FUNCTION_BLOCK GripperCtrl (* Template for a simple Basic Function Block Type *)
  (* Standard: 61499-2 *)
  (* Version 1.0, 2018-07-09, az *)
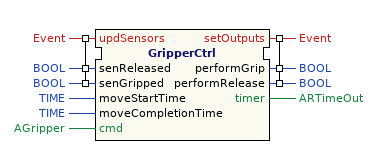
  EVENT_INPUT
    updSensors WITH senReleased, senGripped;
  END_EVENT
  EVENT_OUTPUT
    setOutputs WITH performGrip, performRelease;
  END_EVENT
  VAR_INPUT
    senReleased : BOOL;
    senGripped : BOOL;
    moveStartTime : TIME; (* timeout value till a move should start *)
    moveCompletionTime : TIME; (* timeout till a full movement completes *)
  END_VAR
  VAR_OUTPUT
    performGrip : BOOL;
    performRelease : BOOL;
  END_VAR
  SOCKETS
    cmd : AGripper; (* Command interface for requesting gripper actions *)
  END_SOCKETS
  PLUGS
    timer : ARTimeOut;
  END_PLUGS
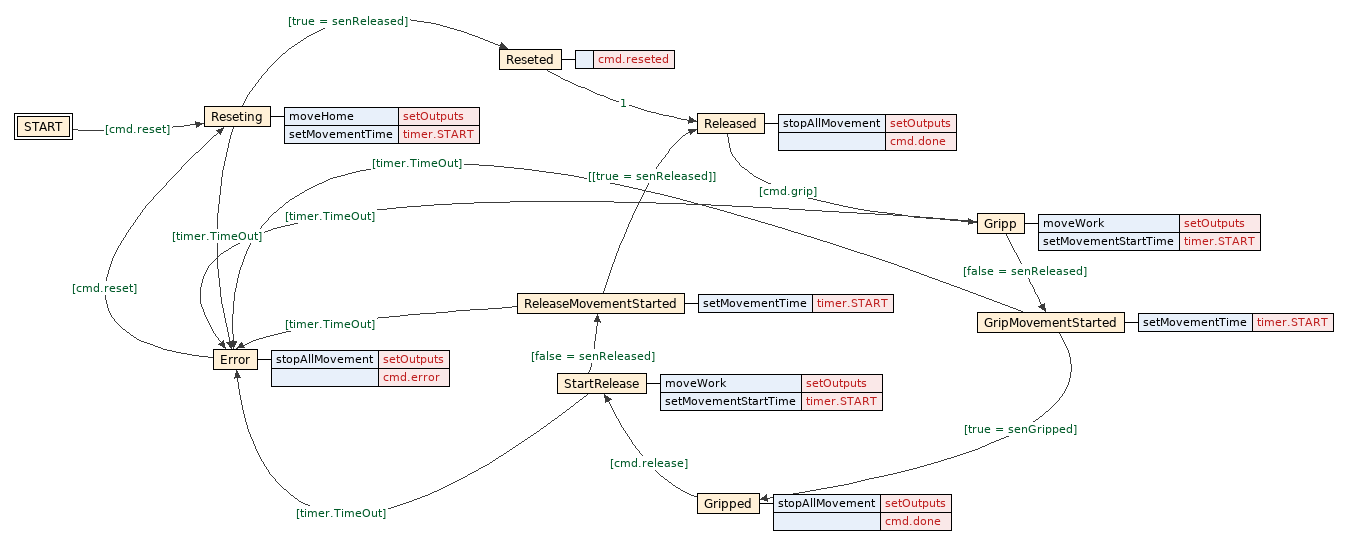
  EC_STATES
    START; (* Initial State *)
    Reseting : moveHome -> setOutputs, setMovementTime -> timer.START; (* Initialization *)
    Error : stopAllMovement -> setOutputs, -> cmd.error;
    Released : stopAllMovement -> setOutputs, -> cmd.done;
    Gripped : stopAllMovement -> setOutputs, -> cmd.done;
    Reseted : -> cmd.reseted;
    Gripp : moveWork -> setOutputs, setMovementStartTime -> timer.START;
    GripMovementStarted : setMovementTime -> timer.START;
    StartRelease : moveWork -> setOutputs, setMovementStartTime -> timer.START;
    ReleaseMovementStarted : setMovementTime -> timer.START;
  END_STATES
  EC_TRANSITIONS
    START TO Reseting := [cmd.reset];
    Error TO Reseting := [cmd.reset];
    Reseted TO Released := 1;
    Reseting TO Reseted := [true = senReleased];
    Reseting TO Error := [timer.TimeOut];
    Gripp TO GripMovementStarted := [false = senReleased];
    GripMovementStarted TO Gripped := [true = senGripped];
    Released TO Gripp := [cmd.grip];
    Gripp TO Error := [timer.TimeOut];
    GripMovementStarted TO Error := [timer.TimeOut];
    Gripped TO StartRelease := [cmd.release];
    StartRelease TO ReleaseMovementStarted := [false = senReleased];
    ReleaseMovementStarted TO Released := [[true = senReleased]];
    ReleaseMovementStarted TO Error := [timer.TimeOut];
    StartRelease TO Error := [timer.TimeOut];
  END_TRANSITIONS
  ALGORITHM moveHome IN ST: (* Initialization algorithm *)
performRelease:= true;
performGrip := false;
  END_ALGORITHM
  ALGORITHM moveWork IN ST: (* Normally executed algorithm *)
performRelease := false;
performGrip := true;
  END_ALGORITHM
  ALGORITHM setMovementStartTime IN ST: (* new algorithm *)
timer.DT := moveStartTime;
  END_ALGORITHM
  ALGORITHM setMovementTime IN ST: (* new algorithm *)
timer.DT := moveCompletionTime;
  END_ALGORITHM
  ALGORITHM stopAllMovement IN ST: (* new algorithm *)
performGrip := false;
performRelease := false;
  END_ALGORITHM
END_FUNCTION_BLOCK
